// SIMATIC S7-200 project (STEP 7-Micro/WIN), CPU 221 REL 01.10

SYMBOL_TABLE USER1
CHE_DO_3         M0.2
CHE_DO_2         M0.1
CHE_DO1          M0.0
ON1              I0.2
ON2              I0.3
ON3              I0.4
OFF              I0.0
DEN              Q0.0
RESET            I0.1
END_SYMBOL_TABLE

ORGANIZATION_BLOCK MAIN:OB1
TITLE=PROGRAM COMMENTS
BEGIN
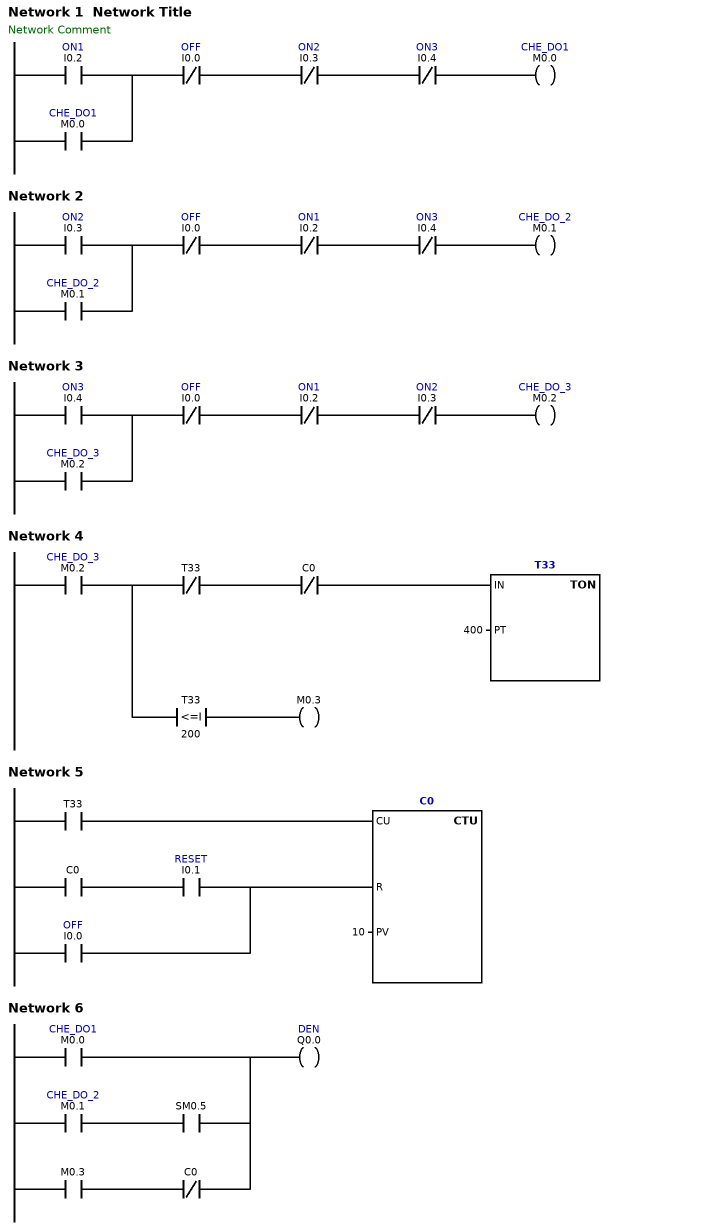
Network 1 // Network Title
// Network Comment
LD     ON1:I0.2
O      CHE_DO1:M0.0
AN     OFF:I0.0
AN     ON2:I0.3
AN     ON3:I0.4
=      CHE_DO1:M0.0
Network 2
LD     ON2:I0.3
O      CHE_DO_2:M0.1
AN     OFF:I0.0
AN     ON1:I0.2
AN     ON3:I0.4
=      CHE_DO_2:M0.1
Network 3
LD     ON3:I0.4
O      CHE_DO_3:M0.2
AN     OFF:I0.0
AN     ON1:I0.2
AN     ON2:I0.3
=      CHE_DO_3:M0.2
Network 4
LD     CHE_DO_3:M0.2
LPS
AN     T33
AN     C0
TON    T33, 400
LPP
AW<=   T33, 200
=      M0.3
Network 5
LD     T33
LD     C0
A      RESET:I0.1
O      OFF:I0.0
CTU    C0, 10
Network 6
LD     CHE_DO1:M0.0
LD     CHE_DO_2:M0.1
A      SM0.5
OLD
LD     M0.3
AN     C0
OLD
=      DEN:Q0.0
END_ORGANIZATION_BLOCK
